FUNCTION_BLOCK OutputCompressor (* Basic Function Block Type *)
  (* Standard: 61499-2 *)
  (* Version 0.0, 6/21/2018, Rediska, nxtControl GmbH, Template *)
  PACKAGE Main;
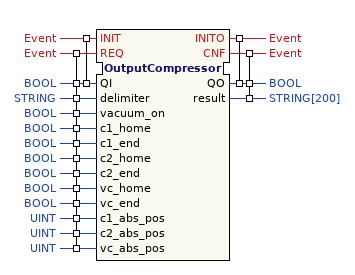
  EVENT_INPUT
    INIT WITH QI; (* Initialization Request *)
    REQ WITH QI, delimiter, vacuum_on, c1_home, c1_end, c2_home, c2_end, vc_home, vc_end, c1_abs_pos, c2_abs_pos, vc_abs_pos; (* Normal Execution Request *)
  END_EVENT
  EVENT_OUTPUT
    INITO WITH QO; (* Initialization Confirm *)
    CNF WITH QO, result; (* Execution Confirmation *)
  END_EVENT
  VAR_INPUT
    QI : BOOL; (* Input event qualifier *)
    delimiter : STRING;
    vacuum_on : BOOL;
    c1_home : BOOL;
    c1_end : BOOL;
    c2_home : BOOL;
    c2_end : BOOL;
    vc_home : BOOL;
    vc_end : BOOL;
    c1_abs_pos : UINT;
    c2_abs_pos : UINT;
    vc_abs_pos : UINT;
  END_VAR
  VAR_OUTPUT
    QO : BOOL; (* Output event qualifier *)
    result : STRING[200];
  END_VAR
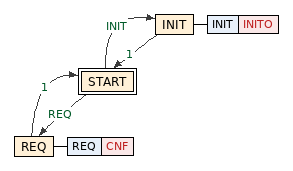
  EC_STATES
    START; (* Initial State *)
    INIT : INIT -> INITO; (* Initialization *)
    REQ : REQ -> CNF; (* Normal execution *)
  END_STATES
  EC_TRANSITIONS
    START TO INIT := INIT;
    INIT TO START := 1;
    START TO REQ := REQ;
    REQ TO START := 1;
  END_TRANSITIONS
  ALGORITHM INIT IN ST: (* Initialization algorithm *)
QO:=TRUE;
  END_ALGORITHM
  ALGORITHM REQ IN ST: (* Normally executed algorithm *)
result :=
CONCAT(
  CONCAT(
    BOOL_TO_STRING(vacuum_on), delimiter,
    BOOL_TO_STRING(c1_home), delimiter,
    BOOL_TO_STRING(c1_end), delimiter
  ),
  CONCAT(
    BOOL_TO_STRING(c2_home), delimiter,
    BOOL_TO_STRING(c2_end), delimiter,
    BOOL_TO_STRING(vc_home), delimiter,
    BOOL_TO_STRING(vc_end), delimiter
  ),
  CONCAT(
    UINT_TO_STRING(c1_abs_pos), delimiter,
    UINT_TO_STRING(c2_abs_pos), delimiter,
    UINT_TO_STRING(vc_abs_pos), delimiter
  ),
  "$N"
);
  END_ALGORITHM
END_FUNCTION_BLOCK
